(* PLC project Sem nome, Desconhecido Sem nome 1 *)
(* stored: creationDateTime 2026-05-26T08:22:23, modificationDateTime 2026-06-09T17:21:49 *)

PROGRAM program0
  VAR
    cancelar AT %IX1.0 : BOOL;
    botao_ligar AT %IX1.1 : BOOL;
    cafe_puro AT %IX1.2 : BOOL;
    cafe_acucar AT %IX1.3 : BOOL;
    cafe_leite_puro AT %IX1.4 : BOOL;
    cafe_leite_acucar AT %IX1.5 : BOOL;
    LED_cancelar AT %QX1.0 : BOOL;
    LED_ligar AT %QX1.1 : BOOL;
  END_VAR
  VAR
    M_start : BOOL;
  END_VAR
  VAR
    sel_cafe_puro AT %QX1.2 : BOOL;
    sel_cafe_acucar AT %QX1.3 : BOOL;
    sel_cafe_leite_puro AT %QX1.4 : BOOL;
    sel_cafe_leite_acucar AT %QX1.5 : BOOL;
    S_nivel_agua AT %IX2.0 : BOOL;
    S_nivel_cafe AT %IX2.1 : BOOL;
    S_nivel_acucar AT %IX2.2 : BOOL;
    S_nivel_leite AT %IX2.3 : BOOL;
    S_xicara AT %IX2.4 : BOOL;
    Valvula_leite AT %QX2.0 : BOOL;  (* 39 *)
    Valvula_agua AT %QX2.1 : BOOL;  (* 41 *)
    Valvula_saida AT %QX2.2 : BOOL;  (* 43 *)
    Dosador_cafe AT %QX2.3 : BOOL;  (* 45 *)
    Dosador_acucar AT %QX2.4 : BOOL;  (* 47 *)
  END_VAR
  VAR
    ingredientes_ok : BOOL;
    T_ingredientes : TON;
    T_mistura : TON;
    T_saida : TON;
    Motor_misturador : BOOL;
  END_VAR
  VAR
    Aquecedor AT %QX1.7 : BOOL;  (* 37 *)
    Buzzer AT %QX1.6 : BOOL;  (* 35 *)
  END_VAR
  VAR  (* added by the conversion: wires and edge detectors of the diagram *)
    R_TRIG1 : R_TRIG;
    R_TRIG2 : R_TRIG;
    R_TRIG3 : R_TRIG;
    R_TRIG4 : R_TRIG;
    R_TRIG5 : R_TRIG;
  END_VAR

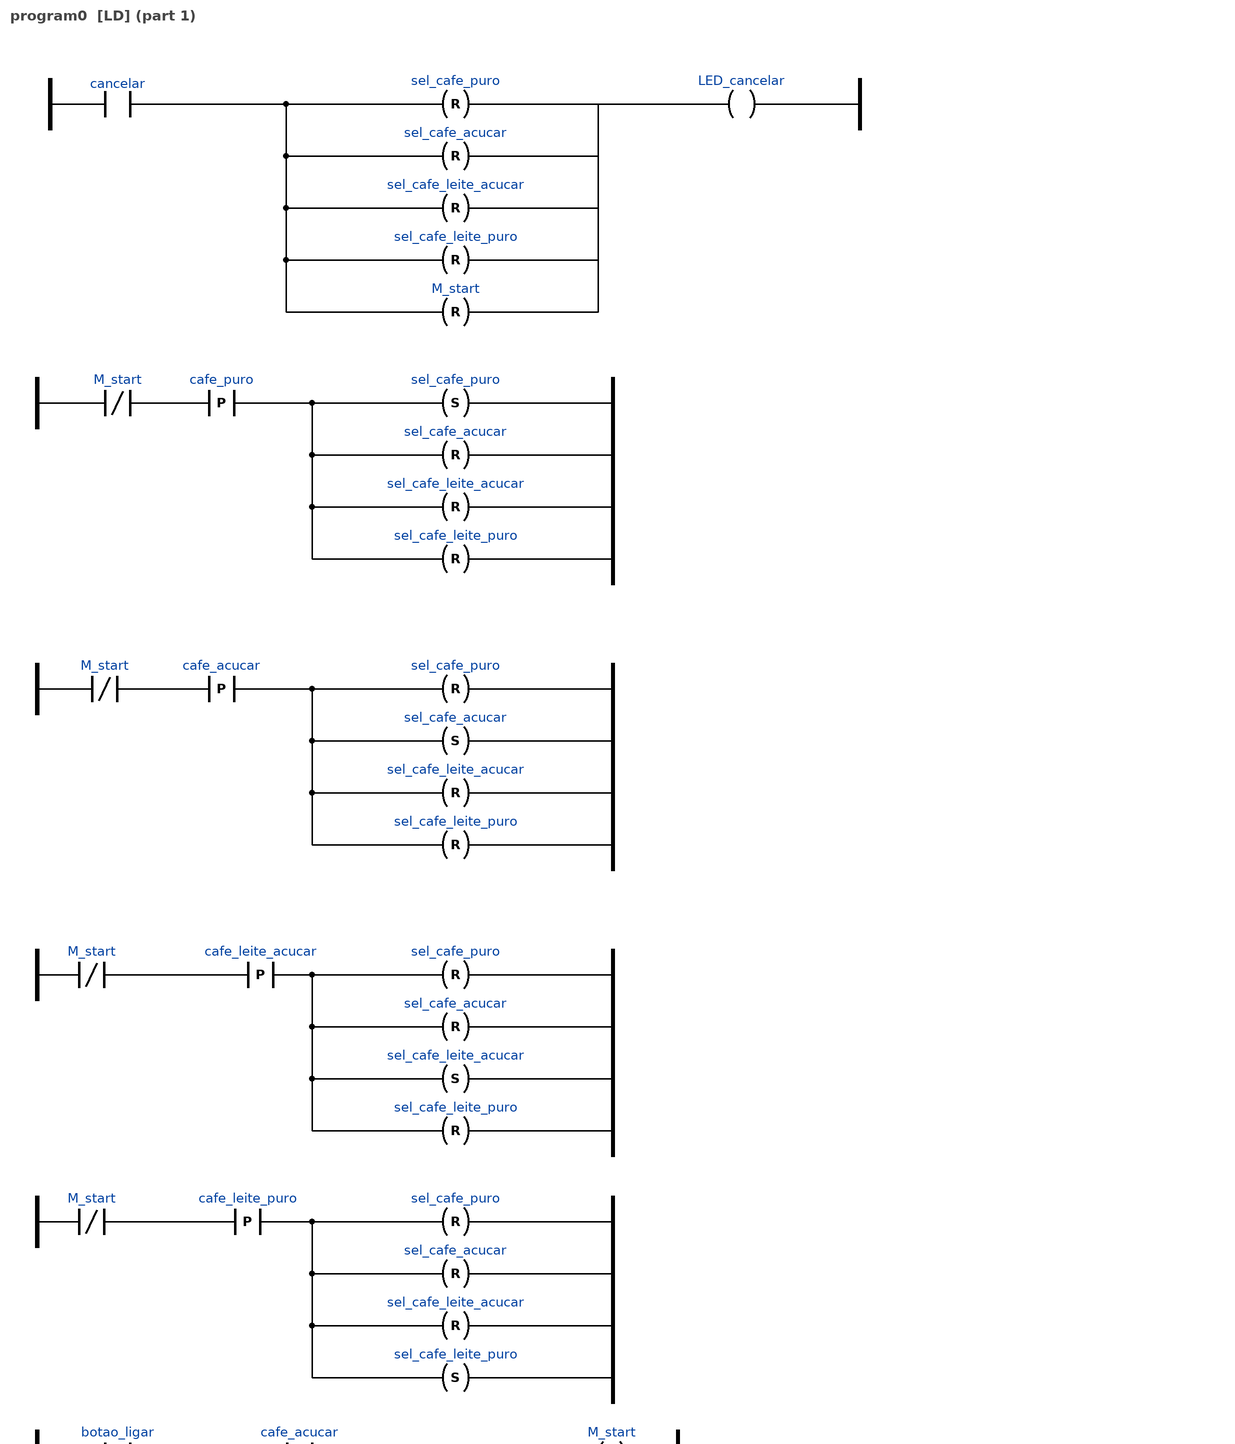
(* LD diagram, written out as Structured Text *)
IF cancelar THEN sel_cafe_puro := FALSE; END_IF;
IF cancelar THEN sel_cafe_leite_puro := FALSE; END_IF;
IF cancelar THEN sel_cafe_leite_acucar := FALSE; END_IF;
IF cancelar THEN sel_cafe_acucar := FALSE; END_IF;
IF cancelar THEN M_start := FALSE; END_IF;
R_TRIG1(CLK := cafe_puro);
IF NOT M_start AND R_TRIG1.Q THEN sel_cafe_puro := TRUE; END_IF;
IF NOT M_start AND R_TRIG1.Q THEN sel_cafe_acucar := FALSE; END_IF;
IF NOT M_start AND R_TRIG1.Q THEN sel_cafe_leite_acucar := FALSE; END_IF;
IF NOT M_start AND R_TRIG1.Q THEN sel_cafe_leite_puro := FALSE; END_IF;
R_TRIG2(CLK := cafe_acucar);
IF NOT M_start AND R_TRIG2.Q THEN sel_cafe_puro := FALSE; END_IF;
IF NOT M_start AND R_TRIG2.Q THEN sel_cafe_acucar := TRUE; END_IF;
IF NOT M_start AND R_TRIG2.Q THEN sel_cafe_leite_acucar := FALSE; END_IF;
IF NOT M_start AND R_TRIG2.Q THEN sel_cafe_leite_puro := FALSE; END_IF;
R_TRIG3(CLK := cafe_leite_acucar);
IF NOT M_start AND R_TRIG3.Q THEN sel_cafe_puro := FALSE; END_IF;
IF NOT M_start AND R_TRIG3.Q THEN sel_cafe_acucar := FALSE; END_IF;
IF NOT M_start AND R_TRIG3.Q THEN sel_cafe_leite_acucar := TRUE; END_IF;
IF NOT M_start AND R_TRIG3.Q THEN sel_cafe_leite_puro := FALSE; END_IF;
R_TRIG4(CLK := cafe_leite_puro);
IF NOT M_start AND R_TRIG4.Q THEN sel_cafe_puro := FALSE; END_IF;
IF NOT M_start AND R_TRIG4.Q THEN sel_cafe_acucar := FALSE; END_IF;
IF NOT M_start AND R_TRIG4.Q THEN sel_cafe_leite_acucar := FALSE; END_IF;
IF NOT M_start AND R_TRIG4.Q THEN sel_cafe_leite_puro := TRUE; END_IF;
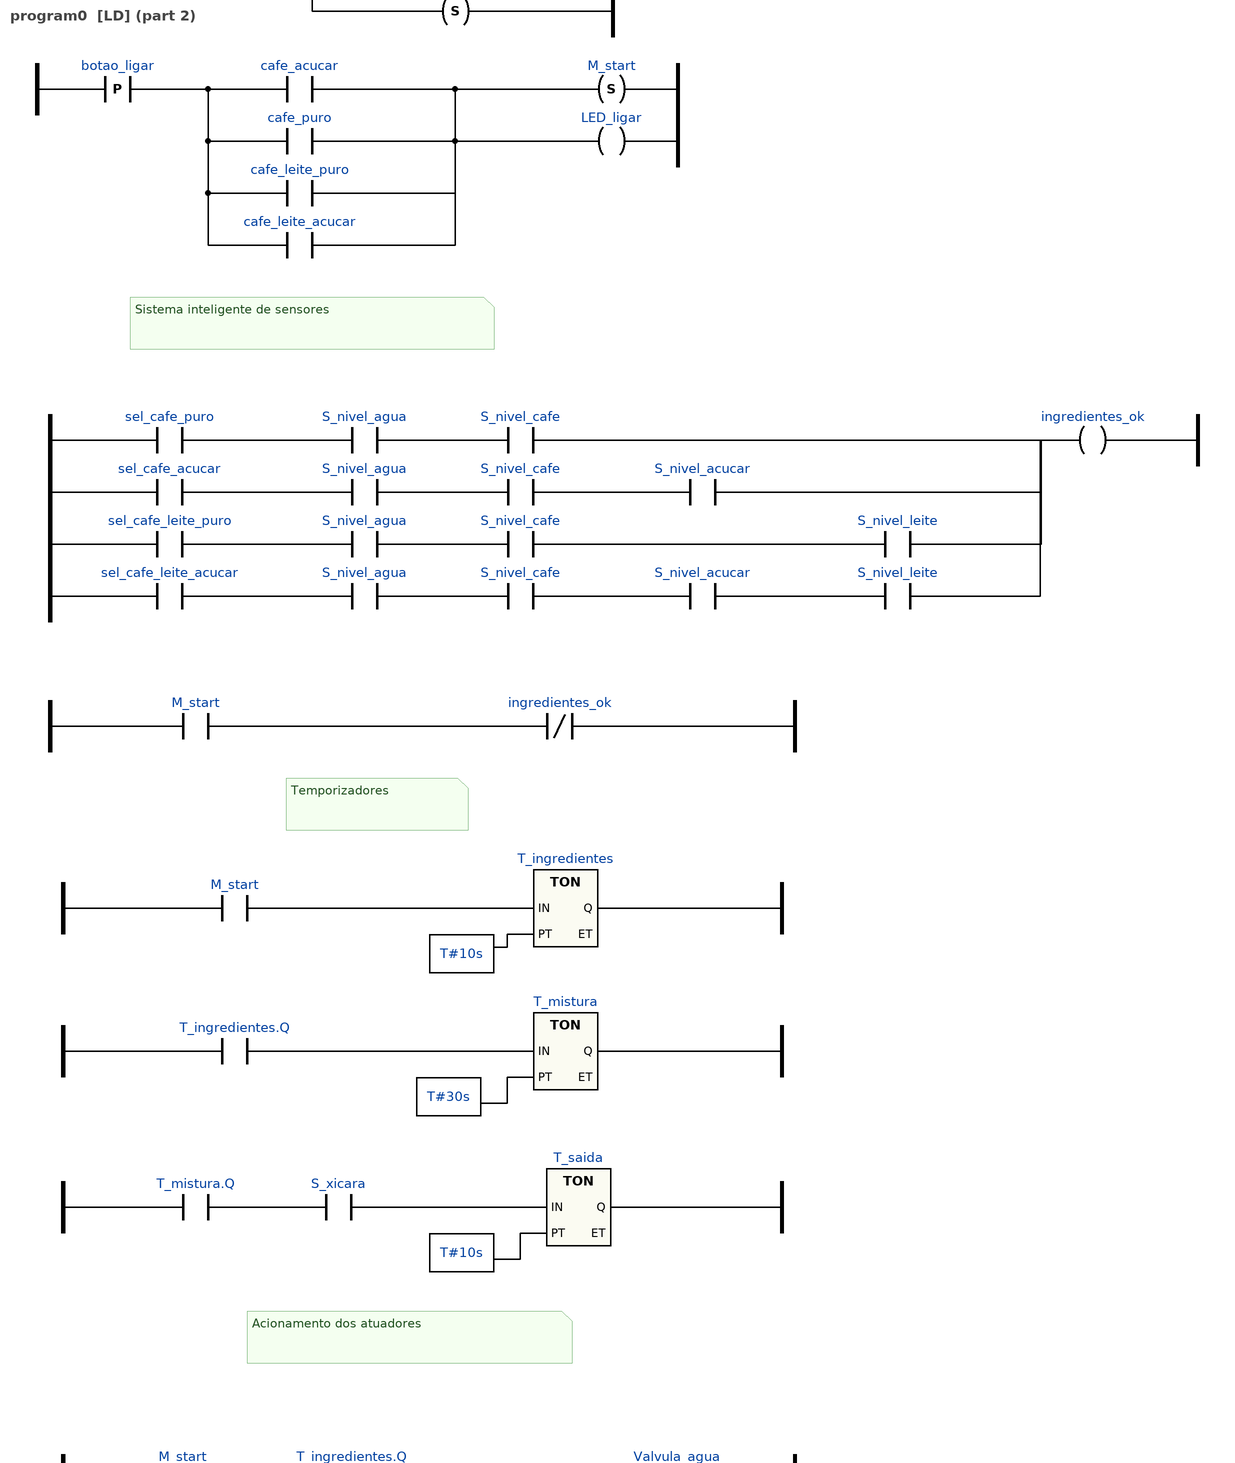
R_TRIG5(CLK := botao_ligar);
IF R_TRIG5.Q AND (cafe_acucar OR cafe_puro OR cafe_leite_puro OR cafe_leite_acucar) THEN M_start := TRUE; END_IF;
(* Sistema inteligente de sensores *)
ingredientes_ok := sel_cafe_puro AND S_nivel_agua AND S_nivel_cafe OR sel_cafe_acucar AND S_nivel_agua AND S_nivel_cafe AND S_nivel_acucar OR sel_cafe_leite_puro AND S_nivel_agua AND S_nivel_cafe AND S_nivel_leite OR sel_cafe_leite_acucar AND S_nivel_agua AND S_nivel_cafe AND S_nivel_acucar AND S_nivel_leite;
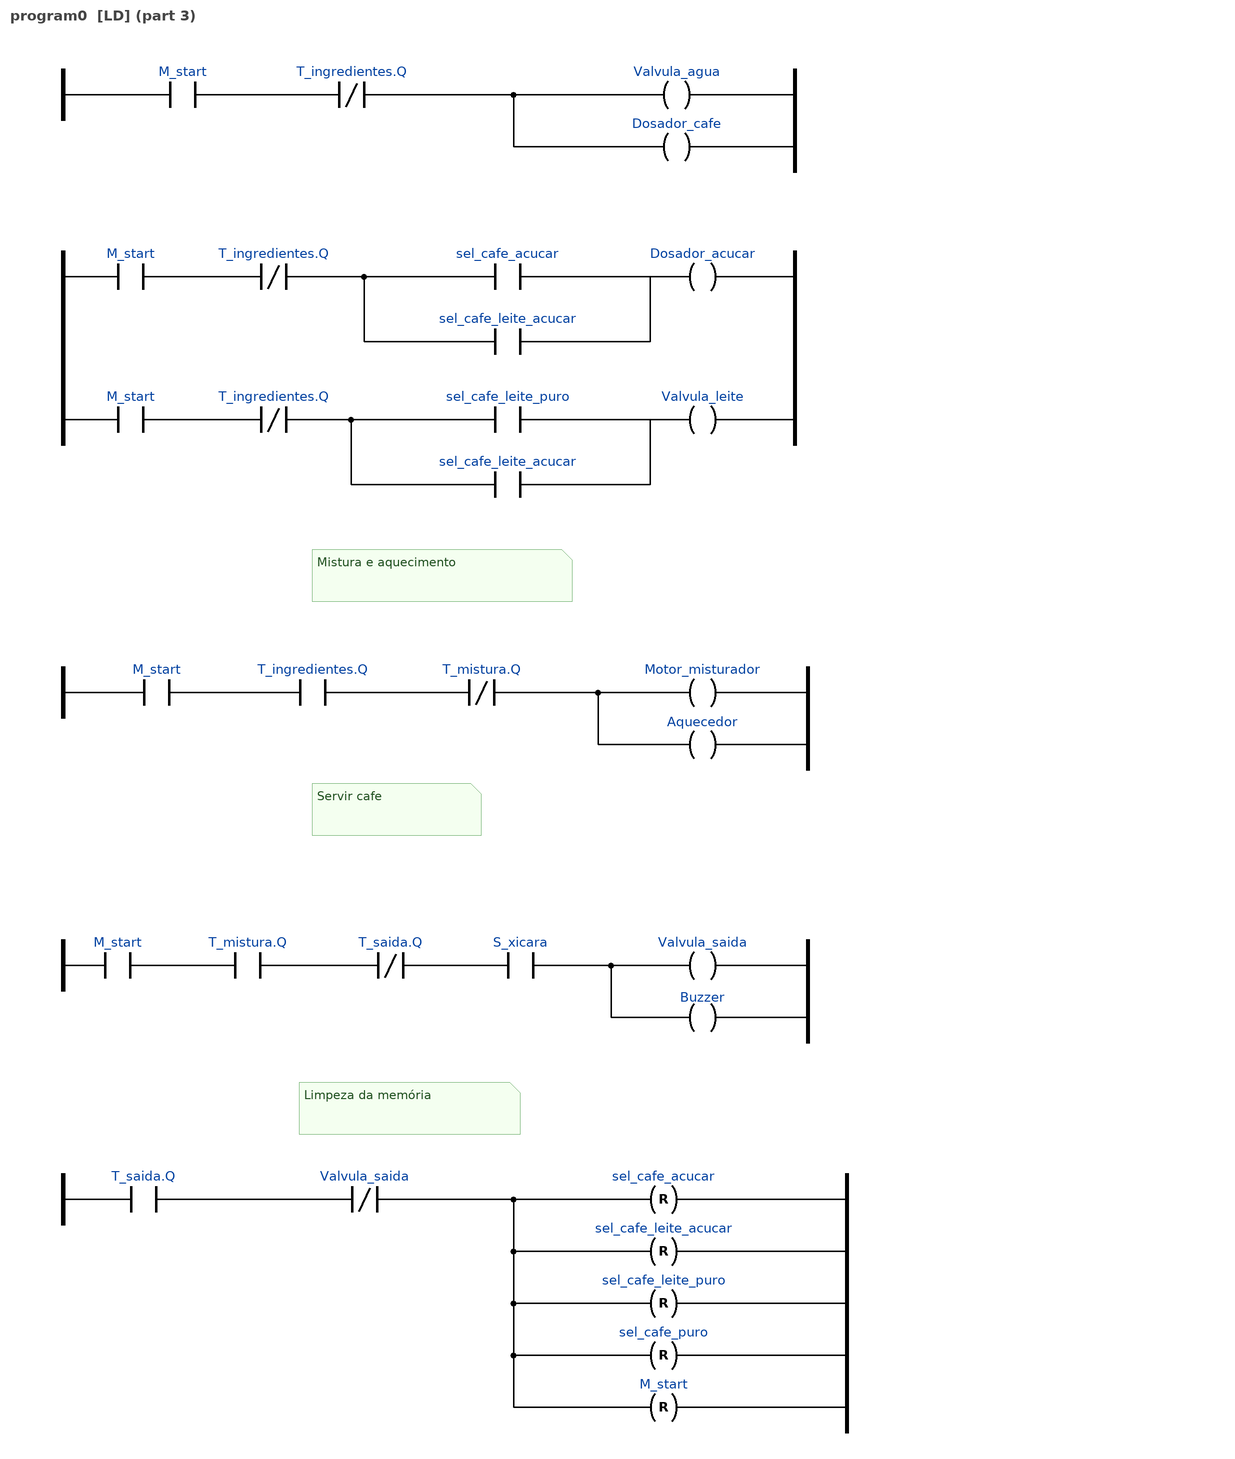
(* Temporizadores *)
(* Acionamento dos atuadores *)
Valvula_agua := M_start AND NOT T_ingredientes.Q;
Dosador_cafe := M_start AND NOT T_ingredientes.Q;
Dosador_acucar := M_start AND NOT T_ingredientes.Q AND (sel_cafe_acucar OR sel_cafe_leite_acucar);
Valvula_leite := M_start AND NOT T_ingredientes.Q AND (sel_cafe_leite_puro OR sel_cafe_leite_acucar);
(* Mistura e aquecimento *)
Motor_misturador := M_start AND T_ingredientes.Q AND NOT T_mistura.Q;
Aquecedor := M_start AND T_ingredientes.Q AND NOT T_mistura.Q;
(* Servir cafe *)
Valvula_saida := M_start AND T_mistura.Q AND NOT T_saida.Q AND S_xicara;
(* Limpeza da memória *)
IF T_saida.Q AND NOT Valvula_saida THEN sel_cafe_acucar := FALSE; END_IF;
IF T_saida.Q AND NOT Valvula_saida THEN sel_cafe_leite_acucar := FALSE; END_IF;
IF T_saida.Q AND NOT Valvula_saida THEN sel_cafe_leite_puro := FALSE; END_IF;
IF T_saida.Q AND NOT Valvula_saida THEN sel_cafe_puro := FALSE; END_IF;
LED_cancelar := cancelar;
LED_ligar := R_TRIG5.Q AND (cafe_puro OR cafe_leite_puro OR cafe_leite_acucar OR cafe_acucar);
Buzzer := M_start AND T_mistura.Q AND NOT T_saida.Q AND S_xicara;
IF T_saida.Q AND NOT Valvula_saida THEN M_start := FALSE; END_IF;
T_ingredientes(IN := M_start, PT := T#10s);
T_mistura(IN := T_ingredientes.Q, PT := T#30s);
T_saida(IN := T_mistura.Q AND S_xicara, PT := T#10s);
(* drawn but not wired to any output: ingredientes_ok, M_start *)
END_PROGRAM

CONFIGURATION Config0
  RESOURCE Res0 ON PLC
    TASK task0(INTERVAL := T#20ms, PRIORITY := 0);
    PROGRAM instance0 WITH task0 : program0;
  END_RESOURCE
END_CONFIGURATION
